ADAPTER OpCdtHMI (* Adapter Interface *)
  (* Standard: 61499-1 *)
  (* Version 0.0, 7/6/2026, Schneider Electric *)
  PACKAGE SE.Nereda;
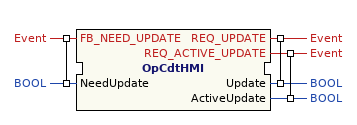
  EVENT_INPUT
    FB_NEED_UPDATE WITH NeedUpdate;
  END_EVENT
  EVENT_OUTPUT
    REQ_UPDATE WITH Update;
    REQ_ACTIVE_UPDATE WITH ActiveUpdate;
  END_EVENT
  VAR_INPUT
    NeedUpdate : BOOL;
  END_VAR
  VAR_OUTPUT
    Update : BOOL;
    ActiveUpdate : BOOL;
  END_VAR
  SERVICE SOCKET/PLUG
    SEQUENCE request_confirm
      SOCKET.REQ(REQD) -> PLUG.REQ(REQD);
      PLUG.CNF(CNFD) -> SOCKET.CNF(CNFD);
    END_SEQUENCE
    SEQUENCE indication_response
      PLUG.IND(INDD) -> SOCKET.IND(INDD);
      SOCKET.RSP(RSPD) -> PLUG.RSP(RSPD);
    END_SEQUENCE
  END_SERVICE
END_ADAPTER
